PROGRAM PRG_LVCP1_Group7
VAR
    // Function Block Instance
    fbContactor: FB_ContactorControl;

    // Contactor 1 IO Structure  
    stContactor_IO: ST_ContactorIO;
    
    // Başlangıç konfigürasyonu için flag
    bContactorInitDone: BOOL := FALSE;
    bCapacitorInitDone: BOOL := FALSE;	
END_VAR



	M_Contactor();
	
	M_Capacitor();

METHOD M_Capacitor : BOOL
VAR
    nGroupIndex : INT;
END_VAR

nGroupIndex := 6;  // Grup 7 için index

IF NOT bCapacitorInitDone THEN
    // Grup 7 değerlerini ata
    GVL_LVCP1.astCompensationGroups[nGroupIndex].rPower := 25.0;
    GVL_LVCP1.astCompensationGroups[nGroupIndex].rVoltage := 450.0;
    GVL_LVCP1.astCompensationGroups[nGroupIndex].nQuantity := 2;
    GVL_LVCP1.astCompensationGroups[nGroupIndex].sTagPrefix := '+EP6-34C1';
    GVL_LVCP1.astCompensationGroups[nGroupIndex].sProductCode := 'ENT.CXD-450-25';
    
    bCapacitorInitDone := TRUE;
END_IF

// Grup 7 aktif durumu
GVL_LVCP1.abGroupActive[nGroupIndex] := stContactor_IO.bFeedback;

M_Capacitor := TRUE;
END_METHOD

METHOD M_Contactor : BOOL
VAR_INPUT
END_VAR
IF NOT bContactorInitDone THEN
    // Konfigürasyon parametreleri
    GVL_LVCP1.stGroup7_ContactorHMI.stConfig.sProjectCode := '+EP6-33K1';
    GVL_LVCP1.stGroup7_ContactorHMI.stConfig.sProductCode := 'SCH LC1G150LSEA';
    GVL_LVCP1.stGroup7_ContactorHMI.stConfig.rRatedCurrent := 150.0;
    GVL_LVCP1.stGroup7_ContactorHMI.stConfig.rRatedVoltage := 1000.0;
    GVL_LVCP1.stGroup7_ContactorHMI.stConfig.nPhaseCount := 3;
    GVL_LVCP1.stGroup7_ContactorHMI.stConfig.tFeedbackDelay := T#500MS;
    GVL_LVCP1.stGroup7_ContactorHMI.stConfig.tWeldedDelay := T#2S;
    GVL_LVCP1.stGroup7_ContactorHMI.stConfig.dwOperationLimit := 100000;
    
    // Başlangıç bakım sayacı
    GVL_LVCP1.stGroup7_ContactorHMI.stStatistics.dwRemainingOperations := GVL_LVCP1.stGroup7_ContactorHMI.stConfig.dwOperationLimit;
    
    bContactorInitDone := TRUE;
END_IF

// Function Block Çağrısı
fbContactor(
    // Fiziksel Girişler
    bFeedback := stContactor_IO.bFeedback,
    bPLCControl := stContactor_IO.bPLCControl,
    
    // Güvenlik Girişleri
    bSafetyLoop := GVL_Alarm.bSafetyLoop,
    bInterlock := FALSE,
    
    // Sistem Girişleri
    bMasterReset := GVL_Alarm.bMasterReset,
    
    // HMI Bağlantısı
    stHMI := GVL_LVCP1.stGroup7_ContactorHMI,
    
    // Fiziksel Çıkış
    bOutput => stContactor_IO.bOutput
);

M_Contactor := TRUE;
END_METHOD

END_PROGRAM

(* stored: Version 1.1.0.1, ProductVersion 3.1.4024.15
   POU PRG_LVCP1_Group7: Id {e595bbdc-e116-48b3-9132-d03c2242d7f6}, SpecialFunc None
   Method M_Capacitor: Id {6ed79b86-ba86-4abc-a5f3-087f105527bb}
   Method M_Contactor: Id {97ac671b-0990-46c6-8c45-f25830252376} *)
